RoboDK station: MoveL_Test-Example.rdk

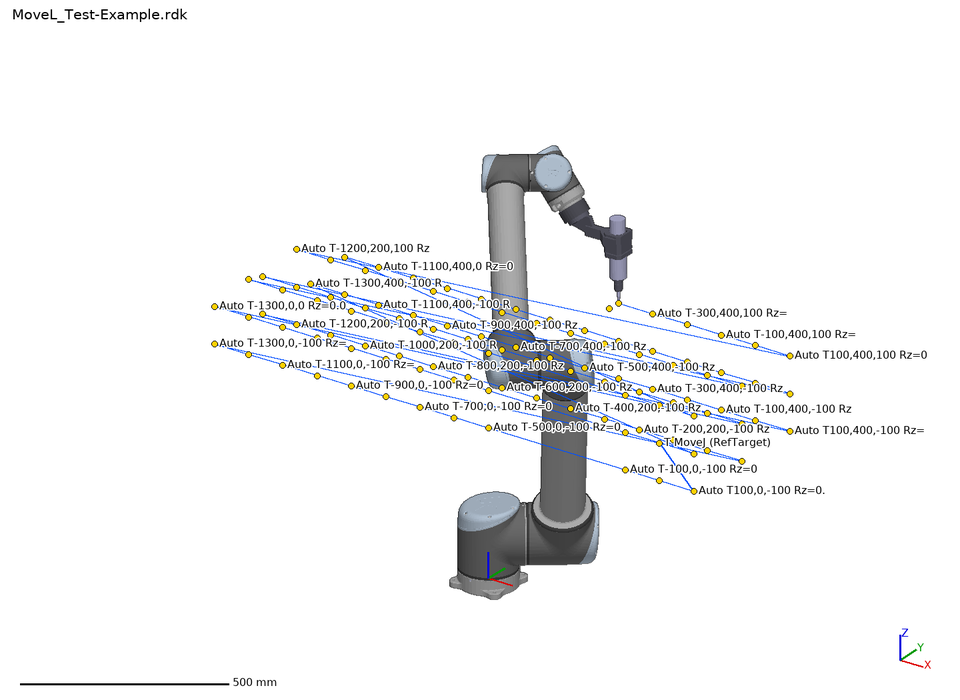
[picture v0: the station drawn from its stored meshes, robots at their saved joint values, targets as dots, program paths as lines]
Station MoveL Test Example. Poses are relative to the parent item; angles as X-Y-Z fixed-axis rotations.
  - frame UR10 Base at (0, 0, 0) mm
    - robot UR10: 6 axes, payload 10 kg, reach 1300 mm, repeatability 0.1 mm, weight 28.9 kg
        modified DH rows (alpha deg, a mm, theta deg, d mm): 0, 0, 0, 118; 90, 0, 180, 0; 0, 612.7, 0, 0; 0, 571.6, 0, 163.9; -90, 0, 0, 115.7; 90, 0, 180, 92.2
        joint limits [-360, -360, -360, -360, -360, -360] to [360, 360, 360, 360, 360, 360]; home [0, -90, 90, 0, 90, 0]; saved at [-232.93, -67.435, 274.582, -143.166, 59.859, -135.81]
      - tool Spindle, TCP at (32, 0, 260) mm, rotated rx 0 ry 39 rz 0 deg, size 157.3 x 72 x 259.9 mm
    - target T MoveJ (RefTarget) (joint target) at (500, 0, 500) mm, rotated rx -180 ry 0 rz 180 deg; joints [32.72, -49.948, 244.302, -70.088, 70.113, 116.533] of UR10
    - target Auto T100,0,-100 Rz=0.0 (Cartesian target) at (600, 0, 400) mm, rotated rx -180 ry 0 rz 180 deg; joints [29.993, -52.418, 242.413, -64.952, 71.664, 114.159] of UR10
    - target Auto T0,0,-100 Rz=0.0 (Cartesian target) at (500, 0, 400) mm, rotated rx -180 ry 0 rz 180 deg; joints [30.628, -51.322, 240.168, -63.977, 71.3, 114.708] of UR10
    - target Auto T-100,0,-100 Rz=0.0 (Cartesian target) at (400, 0, 400) mm, rotated rx -180 ry 0 rz 180 deg; joints [34.134, -47.194, 237.708, -66.681, 69.321, 117.782] of UR10
    - target Auto T-500,0,-100 Rz=0.0 (joint target) at (0, 0, 400) mm, rotated rx -180 ry 0 rz 180 deg; joints [-56.4, -10.264, 237.458, -113.055, 121.613, 40.528] of UR10
    - target Auto T-600,0,-100 Rz=0.0 (Cartesian target) at (-100, 0, 400) mm, rotated rx -180 ry 0 rz 180 deg; joints [-47.719, -6.984, 238.268, -112.702, 117.749, 49.482] of UR10
    - target Auto T-700,0,-100 Rz=0.0 (Cartesian target) at (-200, 0, 400) mm, rotated rx -180 ry 0 rz 180 deg; joints [-38.148, -2.872, 240.544, -115.182, 112.875, 58.6] of UR10
    - target Auto T-800,0,-100 Rz=0.0 (Cartesian target) at (-300, 0, 400) mm, rotated rx -180 ry 0 rz 180 deg; joints [-30.472, 0.89, 244.373, -120.35, 108.611, 65.427] of UR10
    - target Auto T-900,0,-100 Rz=0.0 (Cartesian target) at (-400, 0, 400) mm, rotated rx -180 ry 0 rz 180 deg; joints [-24.776, 3.794, 249.633, -127.102, 105.292, 70.267] of UR10
    - target Auto T-1000,0,-100 Rz=0.0 (Cartesian target) at (-500, 0, 400) mm, rotated rx -180 ry 0 rz 180 deg; joints [-20.545, 5.62, 256.31, -134.757, 102.76, 73.761] of UR10
    - target Auto T-1100,0,-100 Rz=0.0 (Cartesian target) at (-600, 0, 400) mm, rotated rx -180 ry 0 rz 180 deg; joints [-17.371, 6.228, 264.412, -142.941, 100.83, 76.335] of UR10
    - target Auto T-1200,0,-100 Rz=0.0 (Cartesian target) at (-700, 0, 400) mm, rotated rx -180 ry 0 rz 180 deg; joints [-14.936, 5.524, 274.114, -151.597, 99.335, 78.288] of UR10
    - target Auto T-1300,0,-100 Rz=0.0 (joint target) at (-800, 0, 400) mm, rotated rx -180 ry 0 rz 180 deg; joints [-170.536, -123.464, 317.324, -142.476, 95.94, -82.618] of UR10
    - target Auto T100,200,-100 Rz=0.0 (joint target) at (600, 200, 400) mm, rotated rx -180 ry 0 rz 180 deg; joints [-174.973, -8, 268.179, -209.072, 93.161, -86.089] of UR10
    - target Auto T0,200,-100 Rz=0.0 (Cartesian target) at (500, 200, 400) mm, rotated rx -180 ry 0 rz 180 deg; joints [-174.655, -8.426, 266.225, -206.676, 93.361, -85.842] of UR10
    - target Auto T-100,200,-100 Rz=0.0 (Cartesian target) at (400, 200, 400) mm, rotated rx -180 ry 0 rz 180 deg; joints [-173.989, -9.391, 263.026, -202.481, 93.779, -85.322] of UR10
    - target Auto T-200,200,-100 Rz=0.0 (Cartesian target) at (300, 200, 400) mm, rotated rx -180 ry 0 rz 180 deg; joints [-172.819, -11.057, 259.279, -197.001, 94.512, -84.407] of UR10
    - target Auto T-300,200,-100 Rz=0.0 (Cartesian target) at (200, 200, 400) mm, rotated rx -180 ry 0 rz 180 deg; joints [-170.743, -13.502, 255.575, -190.706, 95.81, -82.781] of UR10
    - target Auto T-400,200,-100 Rz=0.0 (Cartesian target) at (100, 200, 400) mm, rotated rx -180 ry 0 rz 180 deg; joints [-166.596, -16.571, 252.36, -184.017, 98.389, -79.508] of UR10
    - target Auto T-500,200,-100 Rz=0.0 (Cartesian target) at (0, 200, 400) mm, rotated rx -180 ry 0 rz 180 deg; joints [-156.735, -19.196, 250.074, -177.525, 104.393, -71.524] of UR10
    - target Auto T-600,200,-100 Rz=0.0 (Cartesian target) at (-100, 200, 400) mm, rotated rx -180 ry 0 rz 180 deg; joints [-133.286, -17.973, 248.772, -169.839, 117.265, -50.474] of UR10
    - target Auto T-700,200,-100 Rz=0.0 (Cartesian target) at (-200, 200, 400) mm, rotated rx -180 ry 0 rz 180 deg; joints [-101.513, -11.12, 247.528, -155.588, 128.073, -14.686] of UR10
    - target Auto T-800,200,-100 Rz=0.0 (Cartesian target) at (-300, 200, 400) mm, rotated rx -180 ry 0 rz 180 deg; joints [-75.875, -3.706, 247.721, -142.837, 127.611, 17.943] of UR10
    - target Auto T-900,200,-100 Rz=0.0 (Cartesian target) at (-400, 200, 400) mm, rotated rx -180 ry 0 rz 180 deg; joints [-58.732, 1.307, 251.142, -139.652, 122.542, 38.003] of UR10
    - target Auto T-1000,200,-100 Rz=0.0 (Cartesian target) at (-500, 200, 400) mm, rotated rx -180 ry 0 rz 180 deg; joints [-47.149, 4.234, 257.231, -142.622, 117.476, 50.045] of UR10
    - target Auto T-1100,200,-100 Rz=0.0 (Cartesian target) at (-600, 200, 400) mm, rotated rx -180 ry 0 rz 180 deg; joints [-39.098, 5.364, 265.316, -148.532, 113.383, 57.727] of UR10
    - target Auto T-1200,200,-100 Rz=0.0 (Cartesian target) at (-700, 200, 400) mm, rotated rx -180 ry 0 rz 180 deg; joints [-33.251, 4.85, 275.228, -155.973, 110.186, 62.999] of UR10
    - target Auto T-1300,200,-100 Rz=0.0 (joint target) at (-800, 200, 400) mm, rotated rx -180 ry 0 rz 180 deg; joints [-182.068, -126.366, 322.127, -144.743, 88.699, -91.607] of UR10
    - target Auto T100,400,-100 Rz=0.0 (Cartesian target) at (600, 400, 400) mm, rotated rx -180 ry 0 rz 180 deg; joints [-187.467, -91.201, 274.784, -132.345, 85.309, -95.816] of UR10
    - target Auto T0,400,-100 Rz=0.0 (Cartesian target) at (500, 400, 400) mm, rotated rx -180 ry 0 rz 180 deg; joints [-195.941, -72.27, 258.631, -134.267, 80.047, -102.516] of UR10
    - target Auto T-100,400,-100 Rz=0.0 (Cartesian target) at (400, 400, 400) mm, rotated rx -180 ry 0 rz 180 deg; joints [-207.138, -62.343, 252.5, -135.935, 73.318, -111.719] of UR10
    - target Auto T-200,400,-100 Rz=0.0 (Cartesian target) at (300, 400, 400) mm, rotated rx -180 ry 0 rz 180 deg; joints [-217.751, -58.601, 250.234, -134.264, 67.338, -121.038] of UR10
    - target Auto T-300,400,-100 Rz=0.0 (Cartesian target) at (200, 400, 400) mm, rotated rx -180 ry 0 rz 180 deg; joints [-224.468, -58.03, 249.531, -131.525, 63.842, -127.338] of UR10
    - target Auto T-400,400,-100 Rz=0.0 (Cartesian target) at (100, 400, 400) mm, rotated rx -180 ry 0 rz 180 deg; joints [-226.716, -58.883, 249.72, -129.876, 62.734, -129.527] of UR10
    - target Auto T-500,400,-100 Rz=0.0 (Cartesian target) at (0, 400, 400) mm, rotated rx -180 ry 0 rz 180 deg; joints [-225.408, -60.583, 250.59, -129.626, 63.375, -128.248] of UR10
    - target Auto T-600,400,-100 Rz=0.0 (Cartesian target) at (-100, 400, 400) mm, rotated rx -180 ry 0 rz 180 deg; joints [-221.986, -63.021, 252.029, -130.052, 65.103, -124.969] of UR10
    - target Auto T-700,400,-100 Rz=0.0 (Cartesian target) at (-200, 400, 400) mm, rotated rx -180 ry 0 rz 180 deg; joints [-217.549, -66.382, 254.122, -130.441, 67.447, -120.853] of UR10
    - target Auto T-800,400,-100 Rz=0.0 (Cartesian target) at (-300, 400, 400) mm, rotated rx -180 ry 0 rz 180 deg; joints [-212.999, -70.68, 256.973, -130.475, 69.956, -116.779] of UR10
    - target Auto T-900,400,-100 Rz=0.0 (Cartesian target) at (-400, 400, 400) mm, rotated rx -180 ry 0 rz 180 deg; joints [-208.775, -75.916, 260.787, -130.238, 72.366, -113.113] of UR10
    - target Auto T-1000,400,-100 Rz=0.0 (Cartesian target) at (-500, 400, 400) mm, rotated rx -180 ry 0 rz 180 deg; joints [-205.128, -81.909, 265.687, -130.024, 74.5, -110.027] of UR10
    - target Auto T-1100,400,-100 Rz=0.0 (Cartesian target) at (-600, 400, 400) mm, rotated rx -180 ry 0 rz 180 deg; joints [-202.051, -88.581, 271.869, -130.179, 76.334, -107.473] of UR10
    - target Auto T-1200,400,-100 Rz=0.0 (Cartesian target) at (-700, 400, 400) mm, rotated rx -180 ry 0 rz 180 deg; joints [-199.509, -95.801, 279.461, -131.014, 77.868, -105.395] of UR10
    - target Auto T-1300,400,-100 Rz=0.0 (Cartesian target) at (-800, 400, 400) mm, rotated rx -180 ry 0 rz 180 deg; joints [-197.394, -103.685, 288.832, -132.843, 79.156, -103.683] of UR10
    - target Auto T100,0,0 Rz=0.0 (joint target) at (600, 0, 500) mm, rotated rx -180 ry 0 rz 180 deg; joints [-203.984, -17.701, 275.35, -204.145, 75.179, -109.072] of UR10
    - target Auto T0,0,0 Rz=0.0 (Cartesian target) at (500, 0, 500) mm, rotated rx -180 ry 0 rz 180 deg; joints [-205.68, -18.246, 273.284, -201.16, 74.174, -110.49] of UR10
    - target Auto T-100,0,0 Rz=0.0 (Cartesian target) at (400, 0, 500) mm, rotated rx -180 ry 0 rz 180 deg; joints [-209.366, -19.461, 269.846, -195.596, 72.024, -113.62] of UR10
    - target Auto T-500,0,0 Rz=0.0 (joint target) at (0, 0, 500) mm, rotated rx -180 ry 0 rz 180 deg; joints [-123.6, -40.434, 255.181, -148.885, 121.613, -40.528] of UR10
    - target Auto T-600,0,0 Rz=0.0 (Cartesian target) at (-100, 0, 500) mm, rotated rx -180 ry 0 rz 180 deg; joints [-132.281, -44.417, 256.356, -150.52, 117.749, -49.482] of UR10
    - target Auto T-700,0,0 Rz=0.0 (Cartesian target) at (-200, 0, 500) mm, rotated rx -180 ry 0 rz 180 deg; joints [-141.852, -50.032, 258.04, -150.499, 112.875, -58.6] of UR10
    - target Auto T-800,0,0 Rz=0.0 (Cartesian target) at (-300, 0, 500) mm, rotated rx -180 ry 0 rz 180 deg; joints [-149.528, -56.42, 260.324, -148.817, 108.611, -65.427] of UR10
    - target Auto T-900,0,0 Rz=0.0 (Cartesian target) at (-400, 0, 500) mm, rotated rx -180 ry 0 rz 180 deg; joints [-155.224, -63.353, 263.488, -146.46, 105.292, -70.267] of UR10
    - target Auto T-1000,0,0 Rz=0.0 (Cartesian target) at (-500, 0, 500) mm, rotated rx -180 ry 0 rz 180 deg; joints [-159.455, -70.8, 267.802, -144.174, 102.76, -73.761] of UR10
    - target Auto T-1100,0,0 Rz=0.0 (Cartesian target) at (-600, 0, 500) mm, rotated rx -180 ry 0 rz 180 deg; joints [-162.629, -78.676, 273.457, -142.48, 100.83, -76.335] of UR10
    - target Auto T-1200,0,0 Rz=0.0 (Cartesian target) at (-700, 0, 500) mm, rotated rx -180 ry 0 rz 180 deg; joints [-165.064, -87.001, 280.692, -141.731, 99.335, -78.288] of UR10
    - target Auto T-1300,0,0 Rz=0.0 (Cartesian target) at (-800, 0, 500) mm, rotated rx -180 ry 0 rz 180 deg; joints [-166.95, -95.769, 289.73, -142.23, 98.169, -79.789] of UR10
    - target Auto T100,200,0 Rz=0.0 (joint target) at (600, 200, 500) mm, rotated rx -180 ry 0 rz 180 deg; joints [-174.973, -17.275, 279.653, -211.27, 93.161, -86.089] of UR10
    - target Auto T0,200,0 Rz=0.0 (Cartesian target) at (500, 200, 500) mm, rotated rx -180 ry 0 rz 180 deg; joints [-174.655, -17.619, 277.677, -208.937, 93.361, -85.842] of UR10
    - target Auto T-100,200,0 Rz=0.0 (Cartesian target) at (400, 200, 500) mm, rotated rx -180 ry 0 rz 180 deg; joints [-173.989, -18.429, 274.474, -204.891, 93.779, -85.322] of UR10
    - target Auto T-200,200,0 Rz=0.0 (Cartesian target) at (300, 200, 500) mm, rotated rx -180 ry 0 rz 180 deg; joints [-172.819, -19.862, 270.766, -199.684, 94.512, -84.407] of UR10
    - target Auto T-300,200,0 Rz=0.0 (Cartesian target) at (200, 200, 500) mm, rotated rx -180 ry 0 rz 180 deg; joints [-170.743, -21.983, 267.146, -193.797, 95.81, -82.781] of UR10
    - target Auto T-400,200,0 Rz=0.0 (Cartesian target) at (100, 200, 500) mm, rotated rx -180 ry 0 rz 180 deg; joints [-166.596, -24.643, 264.037, -187.622, 98.389, -79.508] of UR10
    - target Auto T-500,200,0 Rz=0.0 (Cartesian target) at (0, 200, 500) mm, rotated rx -180 ry 0 rz 180 deg; joints [-156.735, -26.891, 261.814, -181.57, 104.393, -71.524] of UR10
    - target Auto T-600,200,0 Rz=0.0 (Cartesian target) at (-100, 200, 500) mm, rotated rx -180 ry 0 rz 180 deg; joints [-133.286, -25.699, 260.367, -173.707, 117.265, -50.474] of UR10
    - target Auto T-700,200,0 Rz=0.0 (Cartesian target) at (-200, 200, 500) mm, rotated rx -180 ry 0 rz 180 deg; joints [-101.431, -19.378, 258.56, -158.299, 128.086, -14.584] of UR10
    - target Auto T-800,200,0 Rz=0.0 (Cartesian target) at (-300, 200, 500) mm, rotated rx -180 ry 0 rz 180 deg; joints [-76.001, -12.599, 258.057, -144.375, 127.635, 17.786] of UR10
    - target Auto T-900,200,0 Rz=0.0 (Cartesian target) at (-400, 200, 500) mm, rotated rx -180 ry 0 rz 180 deg; joints [-58.794, -7.922, 260.929, -140.247, 122.566, 37.935] of UR10
    - target Auto T-1000,200,0 Rz=0.0 (Cartesian target) at (-500, 200, 500) mm, rotated rx -180 ry 0 rz 180 deg; joints [-47.181, -5.124, 266.638, -142.686, 117.491, 50.014] of UR10
    - target Auto T-1100,200,0 Rz=0.0 (Cartesian target) at (-600, 200, 500) mm, rotated rx -180 ry 0 rz 180 deg; joints [-39.114, -3.998, 274.536, -148.396, 113.392, 57.712] of UR10
    - target Auto T-1200,200,0 Rz=0.0 (Cartesian target) at (-700, 200, 500) mm, rotated rx -180 ry 0 rz 180 deg; joints [-33.273, -4.501, 284.506, -155.906, 110.198, 62.98] of UR10
    - target Auto T-1300,200,0 Rz=0.0 (joint target) at (-800, 200, 500) mm, rotated rx -180 ry 0 rz 180 deg; joints [-182.068, -136.53, 351.44, -163.891, 88.699, -91.607] of UR10
    - target Auto T100,400,0 Rz=0.0 (Cartesian target) at (600, 400, 500) mm, rotated rx -180 ry 0 rz 180 deg; joints [-187.467, -92.638, 286.426, -142.55, 85.309, -95.816] of UR10
    - target Auto T0,400,0 Rz=0.0 (Cartesian target) at (500, 400, 500) mm, rotated rx -180 ry 0 rz 180 deg; joints [-195.941, -74.093, 270.108, -143.92, 80.047, -102.516] of UR10
    - target Auto T-100,400,0 Rz=0.0 (Cartesian target) at (400, 400, 500) mm, rotated rx -180 ry 0 rz 180 deg; joints [-207.138, -64.774, 264.106, -145.11, 73.318, -111.719] of UR10
    - target Auto T-200,400,0 Rz=0.0 (Cartesian target) at (300, 400, 500) mm, rotated rx -180 ry 0 rz 180 deg; joints [-217.751, -61.274, 261.856, -143.212, 67.338, -121.038] of UR10
    - target Auto T-300,400,0 Rz=0.0 (Cartesian target) at (200, 400, 500) mm, rotated rx -180 ry 0 rz 180 deg; joints [-224.468, -60.689, 261.114, -140.449, 63.842, -127.338] of UR10
    - target Auto T-400,400,0 Rz=0.0 (Cartesian target) at (100, 400, 500) mm, rotated rx -180 ry 0 rz 180 deg; joints [-226.716, -61.437, 261.265, -138.867, 62.734, -129.527] of UR10
    - target Auto T-500,400,0 Rz=0.0 (Cartesian target) at (0, 400, 500) mm, rotated rx -180 ry 0 rz 180 deg; joints [-225.408, -63.002, 262.109, -138.726, 63.375, -128.248] of UR10
    - target Auto T-600,400,0 Rz=0.0 (Cartesian target) at (-100, 400, 500) mm, rotated rx -180 ry 0 rz 180 deg; joints [-221.986, -65.275, 263.523, -139.292, 65.103, -124.969] of UR10
    - target Auto T-700,400,0 Rz=0.0 (Cartesian target) at (-200, 400, 500) mm, rotated rx -180 ry 0 rz 180 deg; joints [-217.549, -68.43, 265.582, -139.853, 67.447, -120.853] of UR10
    - target Auto T-800,400,0 Rz=0.0 (Cartesian target) at (-300, 400, 500) mm, rotated rx -180 ry 0 rz 180 deg; joints [-212.999, -72.495, 268.388, -140.075, 69.956, -116.779] of UR10
    - target Auto T-900,400,0 Rz=0.0 (Cartesian target) at (-400, 400, 500) mm, rotated rx -180 ry 0 rz 180 deg; joints [-208.775, -77.505, 272.162, -140.023, 72.366, -113.113] of UR10
    - target Auto T-1000,400,0 Rz=0.0 (Cartesian target) at (-500, 400, 500) mm, rotated rx -180 ry 0 rz 180 deg; joints [-205.128, -83.333, 277.067, -139.98, 74.5, -110.027] of UR10
    - target Auto T-1100,400,0 Rz=0.0 (Cartesian target) at (-600, 400, 500) mm, rotated rx -180 ry 0 rz 180 deg; joints [-202.051, -89.951, 283.365, -140.304, 76.334, -107.473] of UR10
    - target Auto T-1200,400,0 Rz=0.0 (Cartesian target) at (-700, 400, 500) mm, rotated rx -180 ry 0 rz 180 deg; joints [-199.509, -97.29, 291.292, -141.356, 77.868, -105.395] of UR10
    - target Auto T100,0,100 Rz=0.0 (joint target) at (600, 0, 600) mm, rotated rx -180 ry 0 rz 180 deg; joints [-203.984, -27.116, 288.671, -208.052, 75.179, -109.072] of UR10
    - target Auto T0,0,100 Rz=0.0 (Cartesian target) at (500, 0, 600) mm, rotated rx -180 ry 0 rz 180 deg; joints [-205.662, -27.501, 286.521, -205.146, 74.185, -110.475] of UR10
    - target Auto T-100,0,100 Rz=0.0 (Cartesian target) at (400, 0, 600) mm, rotated rx -180 ry 0 rz 180 deg; joints [-209.324, -28.431, 282.956, -199.748, 72.048, -113.584] of UR10
    - target Auto T-500,0,100 Rz=0.0 (joint target) at (0, 0, 600) mm, rotated rx -180 ry 0 rz 180 deg; joints [-123.6, -46.286, 267.994, -155.847, 121.613, -40.528] of UR10
    - target Auto T-600,0,100 Rz=0.0 (Cartesian target) at (-100, 0, 600) mm, rotated rx -180 ry 0 rz 180 deg; joints [-132.281, -49.912, 269.265, -157.934, 117.749, -49.482] of UR10
    - target Auto T-700,0,100 Rz=0.0 (Cartesian target) at (-200, 0, 600) mm, rotated rx -180 ry 0 rz 180 deg; joints [-141.852, -55.013, 271.019, -158.496, 112.875, -58.6] of UR10
    - target Auto T-800,0,100 Rz=0.0 (Cartesian target) at (-300, 0, 600) mm, rotated rx -180 ry 0 rz 180 deg; joints [-149.528, -60.846, 273.33, -157.397, 108.611, -65.427] of UR10
    - target Auto T-900,0,100 Rz=0.0 (Cartesian target) at (-400, 0, 600) mm, rotated rx -180 ry 0 rz 180 deg; joints [-155.224, -67.261, 276.512, -155.576, 105.292, -70.267] of UR10
    - target Auto T-1000,0,100 Rz=0.0 (Cartesian target) at (-500, 0, 600) mm, rotated rx -180 ry 0 rz 180 deg; joints [-159.455, -74.283, 280.886, -153.775, 102.76, -73.761] of UR10
    - target Auto T-1100,0,100 Rz=0.0 (Cartesian target) at (-600, 0, 600) mm, rotated rx -180 ry 0 rz 180 deg; joints [-162.629, -81.894, 286.723, -152.528, 100.83, -76.335] of UR10
    - target Auto T-1200,0,100 Rz=0.0 (Cartesian target) at (-700, 0, 600) mm, rotated rx -180 ry 0 rz 180 deg; joints [-165.064, -90.187, 294.402, -152.256, 99.335, -78.288] of UR10
    - target Auto T100,200,100 Rz=0.0 (joint target) at (600, 200, 600) mm, rotated rx -180 ry 0 rz 180 deg; joints [-174.973, -26.991, 293.308, -215.209, 93.161, -86.089] of UR10
    - target Auto T0,200,100 Rz=0.0 (Cartesian target) at (500, 200, 600) mm, rotated rx -180 ry 0 rz 180 deg; joints [-174.655, -27.193, 291.198, -212.883, 93.361, -85.842] of UR10
    - target Auto T-100,200,100 Rz=0.0 (Cartesian target) at (400, 200, 600) mm, rotated rx -180 ry 0 rz 180 deg; joints [-173.989, -27.763, 287.818, -208.9, 93.779, -85.322] of UR10
    - target Auto T-200,200,100 Rz=0.0 (Cartesian target) at (300, 200, 600) mm, rotated rx -180 ry 0 rz 180 deg; joints [-172.819, -28.888, 283.964, -203.856, 94.512, -84.407] of UR10
    - target Auto T-300,200,100 Rz=0.0 (Cartesian target) at (200, 200, 600) mm, rotated rx -180 ry 0 rz 180 deg; joints [-170.743, -30.642, 280.259, -198.25, 95.81, -82.781] of UR10
    - target Auto T-400,200,100 Rz=0.0 (Cartesian target) at (100, 200, 600) mm, rotated rx -180 ry 0 rz 180 deg; joints [-166.596, -32.893, 277.112, -192.448, 98.389, -79.508] of UR10
    - target Auto T-500,200,100 Rz=0.0 (Cartesian target) at (0, 200, 600) mm, rotated rx -180 ry 0 rz 180 deg; joints [-156.735, -34.787, 274.853, -186.713, 104.393, -71.524] of UR10
    - target Auto T-600,200,100 Rz=0.0 (Cartesian target) at (-100, 200, 600) mm, rotated rx -180 ry 0 rz 180 deg; joints [-133.286, -33.574, 273.207, -178.674, 117.265, -50.474] of UR10
    - target Auto T-700,200,100 Rz=0.0 (Cartesian target) at (-200, 200, 600) mm, rotated rx -180 ry 0 rz 180 deg; joints [-101.431, -27.615, 270.81, -162.313, 128.086, -14.584] of UR10
    - target Auto T-800,200,100 Rz=0.0 (Cartesian target) at (-300, 200, 600) mm, rotated rx -180 ry 0 rz 180 deg; joints [-75.833, -21.217, 269.66, -147.232, 127.603, 17.995] of UR10
    - target Auto T-900,200,100 Rz=0.0 (Cartesian target) at (-400, 200, 600) mm, rotated rx -180 ry 0 rz 180 deg; joints [-58.711, -16.921, 272.135, -142.404, 122.534, 38.026] of UR10
    - target Auto T-1000,200,100 Rz=0.0 (Cartesian target) at (-500, 200, 600) mm, rotated rx -180 ry 0 rz 180 deg; joints [-47.139, -14.401, 277.654, -144.405, 117.471, 50.056] of UR10
    - target Auto T-1100,200,100 Rz=0.0 (Cartesian target) at (-600, 200, 600) mm, rotated rx -180 ry 0 rz 180 deg; joints [-39.092, -13.504, 285.62, -149.967, 113.38, 57.732] of UR10
    - target Auto T-1200,200,100 Rz=0.0 (joint target) at (-700, 200, 600) mm, rotated rx -180 ry 0 rz 180 deg; joints [-182.297, -127.256, 346.415, -168.137, 88.555, -91.785] of UR10
    - target Auto T100,400,100 Rz=0.0 (Cartesian target) at (600, 400, 600) mm, rotated rx -180 ry 0 rz 180 deg; joints [-188.39, -89.161, 293.498, -153.035, 84.732, -96.538] of UR10
    - target Auto T0,400,100 Rz=0.0 (Cartesian target) at (500, 400, 600) mm, rotated rx -180 ry 0 rz 180 deg; joints [-198.059, -73.29, 280.302, -154.604, 78.75, -104.219] of UR10
    - target Auto T-100,400,100 Rz=0.0 (Cartesian target) at (400, 400, 600) mm, rotated rx -180 ry 0 rz 180 deg; joints [-210.41, -66.135, 275.671, -154.465, 71.425, -114.519] of UR10
    - target Auto T-200,400,100 Rz=0.0 (Cartesian target) at (300, 400, 600) mm, rotated rx -180 ry 0 rz 180 deg; joints [-221.296, -63.835, 273.866, -151.348, 65.461, -124.319] of UR10
    - target Auto T-300,400,100 Rz=0.0 (Cartesian target) at (200, 400, 600) mm, rotated rx -180 ry 0 rz 180 deg; joints [-227.541, -63.749, 273.292, -148.206, 62.336, -130.342] of UR10
    - target Auto T-400,400,100 Rz=0.0 (Cartesian target) at (100, 400, 600) mm, rotated rx -180 ry 0 rz 180 deg; joints [-229.012, -64.659, 273.574, -146.89, 61.638, -131.809] of UR10
    - target Auto T-500,400,100 Rz=0.0 (Cartesian target) at (97.3, 364.37, 600) mm, rotated rx -180 ry 0 rz 180 deg; joints [-227.021, -66.222, 274.532, -147.211, 62.586, -129.828] of UR10
  - Python program Make Cube Program (listed below)
  - program AutoCreated (116 instructions, listed below)
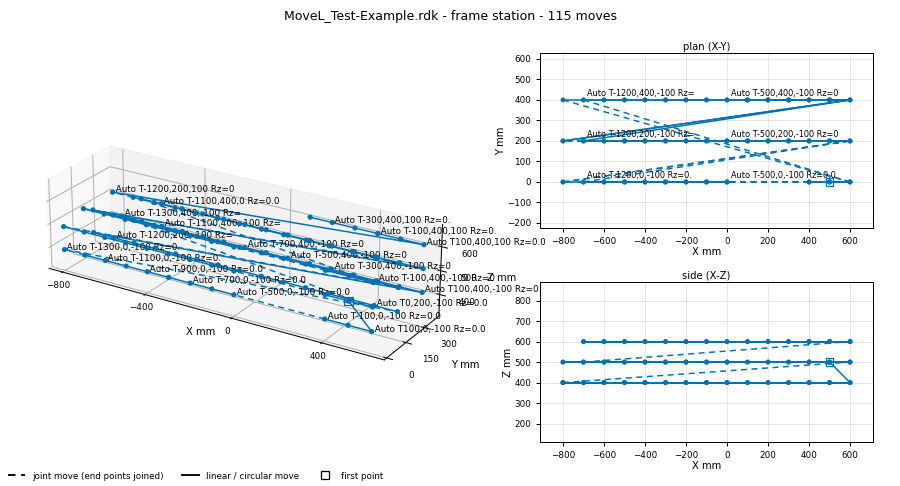
[picture p0: tool path of MoveL_Test-Example.rdk in frame station, 115 of 115 moves have a stored position in this frame; points joined in program order, loops and branches not executed]

--- Python program Make Cube Program ---
from robolink import *    # API to communicate with RoboDK
from robodk import *      # basic matrix operations
from random import uniform # to randomly calculate rz (rotation around the Z axis)

#Start the RoboDK API
RDK = Robolink()

# Run on robot: Force the program to run on the connected robot (same behavior as right clicking the program, then, selecting "Run on Robot")
# RDK.setRunMode(RUNMODE_RUN_ROBOT)

# Get the only robot in the station
robot = RDK.Item('', ITEM_TYPE_ROBOT)

# Get the target reference RefTarget
target_ref = RDK.Item('RefTarget')
# Get the reference position (pose=4x4 matrix of the target with respect to the reference frame)
pose_ref = target_ref.Pose()
startpoint = target_ref.Joints()
config_ref = robot.JointsConfig(startpoint)
tool_pose = robot.Childs()[0].PoseTool()

# Retrieve the degrees of freedom or axes (num_dofs = 6 for a 6 axis robot)
num_dofs = len(robot.JointsHome().list())

# Get the reference frame of the target reference
ref_frame = target_ref.Parent()

def config_equal(config1, config2):
    if config1[0] != config2[0] or config1[1] != config2[1] or config1[2] != config2[2]:
        return False
    return True


# Create a new program
prog = RDK.AddProgram('AutoCreated')

# This should make program generation slightly faster
#prog.ShowInstructions(False)

# Start creating the program or moving the robot:
program_or_robot = prog
program_or_robot.setPoseTool(tool_pose)

program_or_robot.MoveJ(target_ref)
lastjoints = startpoint
rz = 0
ntargets = 0
for tz in range(-100, 101, 100):
    for ty in range(0, 401, 200):
        for tx in range(100, -5001, -250):
            ntargets = ntargets + 1
            # calculate a random rotation around the Z axis of the tool
            #rz = uniform(-20*pi/180, 20*pi/180)

            # Calculate the position of the new target: translate with respect to the robot base and rotate around the tool
            newtarget_pose = transl(tx,ty,tz)*pose_ref*rotz(rz)

            # First, make sure the target is reachable:
            newtarget_joints = robot.SolveIK(newtarget_pose, lastjoints, tool_pose)
            if len(newtarget_joints.tolist()) < num_dofs:
                print('...target not reachable!! Skipping target')
                continue

            # Create a new target:
            newtarget_name = 'Auto T%.0f,%.0f,%.0f Rz=%.1f' % (tx,ty,tz,rz)
            print('Creating target %i: %s' % (ntargets, newtarget_name))
            newtarget = RDK.AddTarget(newtarget_name, ref_frame, robot)

            # At this point, the target is reachable.
            # We have to check if we can do a linear move or not. We have 2 methods:
            can_move_linear = True

            # ------------------------------
            # Validation method 1: check the joints at the destination target
            # and make sure we have the same configuration
            # A quick way to validate (it may not be perfect if robot joints can move more than 1 turn)
            # To improve this method we would have to check configurations on all possible solutions
            # from the inverse kinematics, using SolveIK_All()
            if False:
                target_joints_config = robot.JointsConfig(newtarget_joints)
                if not config_equal(config_ref, target_joints_config):
                    # We can't do a linear movement
                    can_move_linear = False
                    print("Warning! configuration is not the same as the reference target! Linear move will not be possible")

                    # update the reference configuration to the new one
                    config_ref = target_joints_config
            # -------------------------------



            # -------------------------------
            # Validation method 2: use the robot.MoveL_Test option to check if the robot can make a linear movement
            # This method is more robust and should provide a 100% accurate result but it may take more time
            # robot.MoveL_Test can also take collisions into account if collision checking is activated
            issues = robot.MoveL_Test(lastjoints, newtarget_pose)
            can_move_linear = (issues == 0)
            # We can retrieve the final joint position by retrieving the robot joints
            if can_move_linear:
                newtarget_joints = robot.Joints()

            # ---------------------------------

            if can_move_linear:
                # All good, we don't need to modify the target.
                # However, we could set the joints in the target as this may allow us to retrieve the robot configuration if we ever need it
                newtarget.setAsCartesianTarget() # default behavior
                newtarget.setJoints(newtarget_joints)
                # It is important to have setPose after setJoints as it may recalculate the joints to match the target
                newtarget.setPose(newtarget_pose)

                # Add the linear movement
                program_or_robot.MoveL(newtarget)

            else:
                print(newtarget_joints)
                # Make sure we have a joint target and a joint movement
                newtarget.setAsJointTarget() # default behavior

                # Setting the pose for a joint target is not important unless we want to retrieve the pose later
                # or we want to use the Cartesian coordinates for post processing
                newtarget.setPose(newtarget_pose)

                # Make sure we set the joints after the pose for a joint taget as it may recalculate the pose
                newtarget.setJoints(newtarget_joints)

                # Add the joint movement
                program_or_robot.MoveJ(newtarget)


            # Remember the joint poisition of the last movement
            lastjoints = newtarget_joints

# Showing the instructions at the end is faster:
prog.ShowInstructions(True)

# Hiding the targets is cleaner and more difficult to accidentaly move a target
#prog.ShowTargets(False)

print('Program done with %i targets' % ntargets)

--- program AutoCreated (robot UR10) ---
  Set Tool at (32, 0, 260) mm, rotated rx 0 ry 39 rz 0 deg
  MoveJ (T MoveJ (RefTarget))
  MoveL (Auto T100,0,-100 Rz=0.0)
  MoveL (Auto T0,0,-100 Rz=0.0)
  MoveL (Auto T-100,0,-100 Rz=0.0)
  MoveJ (Auto T-500,0,-100 Rz=0.0)
  MoveL (Auto T-600,0,-100 Rz=0.0)
  MoveL (Auto T-700,0,-100 Rz=0.0)
  MoveL (Auto T-800,0,-100 Rz=0.0)
  MoveL (Auto T-900,0,-100 Rz=0.0)
  MoveL (Auto T-1000,0,-100 Rz=0.0)
  MoveL (Auto T-1100,0,-100 Rz=0.0)
  MoveL (Auto T-1200,0,-100 Rz=0.0)
  MoveJ (Auto T-1300,0,-100 Rz=0.0)
  MoveJ (Auto T100,200,-100 Rz=0.0)
  MoveL (Auto T0,200,-100 Rz=0.0)
  MoveL (Auto T-100,200,-100 Rz=0.0)
  MoveL (Auto T-200,200,-100 Rz=0.0)
  MoveL (Auto T-300,200,-100 Rz=0.0)
  MoveL (Auto T-400,200,-100 Rz=0.0)
  MoveL (Auto T-500,200,-100 Rz=0.0)
  MoveL (Auto T-600,200,-100 Rz=0.0)
  MoveL (Auto T-700,200,-100 Rz=0.0)
  MoveL (Auto T-800,200,-100 Rz=0.0)
  MoveL (Auto T-900,200,-100 Rz=0.0)
  MoveL (Auto T-1000,200,-100 Rz=0.0)
  MoveL (Auto T-1100,200,-100 Rz=0.0)
  MoveL (Auto T-1200,200,-100 Rz=0.0)
  MoveJ (Auto T-1300,200,-100 Rz=0.0)
  MoveL (Auto T100,400,-100 Rz=0.0)
  MoveL (Auto T0,400,-100 Rz=0.0)
  MoveL (Auto T-100,400,-100 Rz=0.0)
  MoveL (Auto T-200,400,-100 Rz=0.0)
  MoveL (Auto T-300,400,-100 Rz=0.0)
  MoveL (Auto T-400,400,-100 Rz=0.0)
  MoveL (Auto T-500,400,-100 Rz=0.0)
  MoveL (Auto T-600,400,-100 Rz=0.0)
  MoveL (Auto T-700,400,-100 Rz=0.0)
  MoveL (Auto T-800,400,-100 Rz=0.0)
  MoveL (Auto T-900,400,-100 Rz=0.0)
  MoveL (Auto T-1000,400,-100 Rz=0.0)
  MoveL (Auto T-1100,400,-100 Rz=0.0)
  MoveL (Auto T-1200,400,-100 Rz=0.0)
  MoveL (Auto T-1300,400,-100 Rz=0.0)
  MoveJ (Auto T100,0,0 Rz=0.0)
  MoveL (Auto T0,0,0 Rz=0.0)
  MoveL (Auto T-100,0,0 Rz=0.0)
  MoveJ (Auto T-500,0,0 Rz=0.0)
  MoveL (Auto T-600,0,0 Rz=0.0)
  MoveL (Auto T-700,0,0 Rz=0.0)
  MoveL (Auto T-800,0,0 Rz=0.0)
  MoveL (Auto T-900,0,0 Rz=0.0)
  MoveL (Auto T-1000,0,0 Rz=0.0)
  MoveL (Auto T-1100,0,0 Rz=0.0)
  MoveL (Auto T-1200,0,0 Rz=0.0)
  MoveL (Auto T-1300,0,0 Rz=0.0)
  MoveJ (Auto T100,200,0 Rz=0.0)
  MoveL (Auto T0,200,0 Rz=0.0)
  MoveL (Auto T-100,200,0 Rz=0.0)
  MoveL (Auto T-200,200,0 Rz=0.0)
  MoveL (Auto T-300,200,0 Rz=0.0)
  MoveL (Auto T-400,200,0 Rz=0.0)
  MoveL (Auto T-500,200,0 Rz=0.0)
  MoveL (Auto T-600,200,0 Rz=0.0)
  MoveL (Auto T-700,200,0 Rz=0.0)
  MoveL (Auto T-800,200,0 Rz=0.0)
  MoveL (Auto T-900,200,0 Rz=0.0)
  MoveL (Auto T-1000,200,0 Rz=0.0)
  MoveL (Auto T-1100,200,0 Rz=0.0)
  MoveL (Auto T-1200,200,0 Rz=0.0)
  MoveJ (Auto T-1300,200,0 Rz=0.0)
  MoveL (Auto T100,400,0 Rz=0.0)
  MoveL (Auto T0,400,0 Rz=0.0)
  MoveL (Auto T-100,400,0 Rz=0.0)
  MoveL (Auto T-200,400,0 Rz=0.0)
  MoveL (Auto T-300,400,0 Rz=0.0)
  MoveL (Auto T-400,400,0 Rz=0.0)
  MoveL (Auto T-500,400,0 Rz=0.0)
  MoveL (Auto T-600,400,0 Rz=0.0)
  MoveL (Auto T-700,400,0 Rz=0.0)
  MoveL (Auto T-800,400,0 Rz=0.0)
  MoveL (Auto T-900,400,0 Rz=0.0)
  MoveL (Auto T-1000,400,0 Rz=0.0)
  MoveL (Auto T-1100,400,0 Rz=0.0)
  MoveL (Auto T-1200,400,0 Rz=0.0)
  MoveJ (Auto T100,0,100 Rz=0.0)
  MoveL (Auto T0,0,100 Rz=0.0)
  MoveL (Auto T-100,0,100 Rz=0.0)
  MoveJ (Auto T-500,0,100 Rz=0.0)
  MoveL (Auto T-600,0,100 Rz=0.0)
  MoveL (Auto T-700,0,100 Rz=0.0)
  MoveL (Auto T-800,0,100 Rz=0.0)
  MoveL (Auto T-900,0,100 Rz=0.0)
  MoveL (Auto T-1000,0,100 Rz=0.0)
  MoveL (Auto T-1100,0,100 Rz=0.0)
  MoveL (Auto T-1200,0,100 Rz=0.0)
  MoveJ (Auto T100,200,100 Rz=0.0)
  MoveL (Auto T0,200,100 Rz=0.0)
  MoveL (Auto T-100,200,100 Rz=0.0)
  MoveL (Auto T-200,200,100 Rz=0.0)
  MoveL (Auto T-300,200,100 Rz=0.0)
  MoveL (Auto T-400,200,100 Rz=0.0)
  MoveL (Auto T-500,200,100 Rz=0.0)
  MoveL (Auto T-600,200,100 Rz=0.0)
  MoveL (Auto T-700,200,100 Rz=0.0)
  MoveL (Auto T-800,200,100 Rz=0.0)
  MoveL (Auto T-900,200,100 Rz=0.0)
  MoveL (Auto T-1000,200,100 Rz=0.0)
  MoveL (Auto T-1100,200,100 Rz=0.0)
  MoveJ (Auto T-1200,200,100 Rz=0.0)
  MoveL (Auto T100,400,100 Rz=0.0)
  MoveL (Auto T0,400,100 Rz=0.0)
  MoveL (Auto T-100,400,100 Rz=0.0)
  MoveL (Auto T-200,400,100 Rz=0.0)
  MoveL (Auto T-300,400,100 Rz=0.0)
  MoveL (Auto T-400,400,100 Rz=0.0)
